TYPE ST_VariableLink :
STRUCT
	SourceAddress : PVOID;
	TargetAddress : PVOID;
	SourceSize : UDINT;
	TargetSize : UDINT;
	SourceDataType : E_ConfigDataType;
	TargetDataType : E_ConfigDataType;
	Phase : E_LinkPhase;
	HasTransform : BOOL;
	Scale : LREAL;
	Offset : LREAL;
END_STRUCT
END_TYPE

(* stored: Version 1.1.0.1, ProductVersion 3.1.4026.18
   DUT ST_VariableLink: Id {a782d317-ed91-4129-b2a5-7c267b1556fe} *)
